{attribute 'linkalways'}
{attribute 'some_made_up_key':='some_made_up_value'}
FUNCTION_BLOCK AttributeTest
VAR
END_VAR

END_FUNCTION_BLOCK

(* stored: Version 1.1.0.1, ProductVersion 3.1.4024.13
   POU AttributeTest: Id {957860c0-06d0-4a53-9b3d-b3dab5789371}, SpecialFunc None *)
